(* PLC project Unnamed, Unknown Unnamed 1 *)
(* stored: creationDateTime 2019-08-06T14:23:42, modificationDateTime 2019-08-09T11:20:07 *)

PROGRAM program0
  VAR
    LocalVar0 : DINT;
  END_VAR

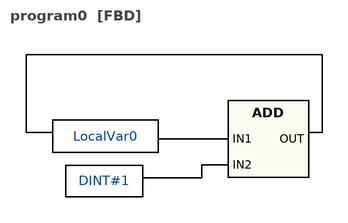
(* FBD diagram, written out as Structured Text *)
LocalVar0 := LocalVar0 + DINT#1;
END_PROGRAM

CONFIGURATION config
  RESOURCE resource1 ON PLC
    TASK task0(INTERVAL := T#20ms, PRIORITY := 0);
    PROGRAM instance0 WITH task0 : program0;
  END_RESOURCE
END_CONFIGURATION
